Staubli VAL3: listempty.pgx

public program listEmpty()
  local num i
  local num l_nSize
begin
  //-----------------------------------------------------------------------
  //Header begin
  //Description of program
  //  Delete all the elements of the list (sItems).
  //
  //Example
  //  call listEmpty()
  //
  //History
  //  Creation : 28-04-08 - f.Rob
  //Header end
  //-----------------------------------------------------------------------
  l_nSize=size(sItems)-1
  for i=0 to l_nSize
    if i>0
      //Destroy all elements of sItems
      delete(sItems[0])
      //Destroy all elements of bReadWrite
      delete(bReadWrite[0])
    endIf
  endFor
  sItems=""
end
